FUNCTION_BLOCK Test_TStreamAdd_Read_STRING EXTENDS T_UnitTestBase
VAR
    Stream     : T_Stream(StreamLength := 2);
    ArgType    : E_ArgTypeId := E_ArgTypeId.Type_STRING;
    TestString : STRING      := '111111111 222222222 333333333 444444444 555555555 666666666 777777777 888888888 ';
END_VAR

{attribute 'analysis' := '-33'} // inhibit unused variable warning
METHOD RunTest
IF Retest THEN
    SUPER^.Init();
END_IF

IF TestCompleted THEN
    RETURN;
END_IF

F_Inc(CycleCount);
IF CycleCount > 1000 THEN
    Fail(Message := 'Timeout');
END_IF

Stream.Init(2);

// add a STRING...
Stream.SetNextArgTypeId(ArgType);
Stream.Add_STRING(TestString);

Stream.SetReadPosition(0);

// check next arg type is correct...
AssertEquals_INT(Expected     := ArgType,
                           Actual       := Stream.GetNextArgTypeId(),
                           Message := 'Stream.GetNextArgTypeId()');

// check next value...	
AssertEquals_STRING(Expected     := TestString,
                              Actual       := Stream.Read_STRING(),
                              Message := 'Stream.Read_STRING()');

// check we are at the end of the stream..							
AssertEquals_UDINT(Expected     := Stream.StreamLength,
                             Actual       := Stream.ReadPosition,
                             Message := 'Stream.ReadPosition');

TestCompleted := TRUE;
END_METHOD

END_FUNCTION_BLOCK

(* stored: Version 1.1.0.1, ProductVersion 3.1.4024.15
   POU Test_TStreamAdd_Read_STRING: Id {2e1a9193-2c9c-4120-b4b0-ca0f5d5f8274}, SpecialFunc None
   Method RunTest: Id {8c89a821-d26d-4065-bb5d-6d06583b73f6} *)
